FUNCTION_BLOCK FB_Hmi_Led
VAR_INPUT
END_VAR
VAR_OUTPUT
END_VAR
VAR
END_VAR

END_FUNCTION_BLOCK

(* stored: Version 1.1.0.1, ProductVersion 3.1.4024.10
   POU FB_Hmi_Led: Id {629fea12-c436-4ed1-9312-b78a6f33c585}, SpecialFunc None *)
